// TIA Portal V17 export
// export: Created 2025-04-09T07:53:25.722931Z, ExportSetting WithDefaults, DisplayName Totally Integrated Automation Portal, DisplayVersion V17, DisplayName TIA Portal Openness, DisplayVersion V17, DisplayName TIA Portal Version Control Interface, DisplayVersion V17, DisplayName STEP 7 Professional, DisplayVersion V17, DisplayName STEP 7 Safety, DisplayVersion V17, DisplayName WinCC Advanced, DisplayVersion V17
DATA_BLOCK "Raktario"   // DB1
{ S7_Optimized_Access := 'TRUE' }
VERSION : 0.1
// stored: AutoNumber true, DBAccessibleFromOPCUA true, IsOnlyStoredInLoadMemory false, IsRetainMemResEnabled false, IsWriteProtectedInAS false, MemoryReserve 100
   VAR
      Input : Struct
         START : Bool;
         STOP : Bool;
         MODE : Bool;
         PRES : Bool;
         REQ_A : Bool;
         REQ_B : Bool;
         COL_A : Bool;
         COL_B : Bool;
         RAD_OFF : Bool;
         RAD_ON : Bool;
         AX_RDY : Bool;
         ANG_RDY : Bool;
      END_STRUCT;
      Internal : Struct
         Bekeres : Struct
            pirosker : Bool;
            feketeker : Bool;
            feherker : Bool;
            nincsker : Bool;
         END_STRUCT;
         Szinerzekelo : Struct
            nincs : Bool;
            piros : Bool;
            fekete : Bool;
            feher : Bool;
         END_STRUCT;
         Hetszegmens : Struct
            Sotet : Bool;
            "1" : Bool;
            "2" : Bool;
            "3" : Bool;
            "4" : Bool;
            P : Bool;
            "E" : Bool;
            F : Bool;
         END_STRUCT;
         Pozicio : Struct
            "A" : Bool;
            "B" : Bool;
            C : Bool;
            D : Bool;
            "E" : Bool;
            F : Bool;
            G : Bool;
            H : Bool;
            "1" : Bool;
            "2" : Bool;
            "3" : Bool;
            "4" : Bool;
            "5" : Bool;
            "6" : Bool;
            "7" : Bool;
            "8" : Bool;
            angstart : Bool;
            angstop : Bool;
            axstart : Bool;
            axstop : Bool;
            mempiros : Byte := 16#38;
            memfekete : Byte := 16#38;
            memezust : Byte := 16#38;
         END_STRUCT;
      END_STRUCT;
      Output : Struct
         RUN : Bool;
         STATUS : Bool;
         ERROR : Bool;
         SS_A : Bool;
         SS_B : Bool;
         SS_C : Bool;
         RAD : Bool;
         GRIP : Bool;
         POS_A : Bool;
         POS_B : Bool;
         POS_C : Bool;
         AX_ST : Bool;
         ANG_ST : Bool;
         COLOR : Bool;
      END_STRUCT;
   END_VAR
BEGIN
END_DATA_BLOCK
